INTERFACE I_LREAL EXTENDS I_Datatype

{warning disable C5410}
PROPERTY PUBLIC Value : REFERENCE TO LREAL
{warning restore C5410}
GET
END_GET
END_PROPERTY

END_INTERFACE

(* stored: Version 1.1.0.1, ProductVersion 3.1.4024.15
   Itf I_LREAL: Id {240ec6c4-cec3-0089-1328-49e6df1d5728}
   Property Value: Id {d2f69e8a-bf83-0a22-0ffe-c3959cabad5a}
   Get Get: Id {4ae2590c-6b39-05b0-1bf1-c206cecc4ea8} *)
